# EPICS substitutions: bkhApp/Db/bkh09.substitutions
file bkhBo.db
{
pattern	{ N,       MOD,  PORT, OFF}
	{ 1, 2114-$(M), A2114,   0}
	{ 2, 2114-$(M), A2114,   1}
	{ 3, 2114-$(M), A2114,   2}
	{ 4, 2114-$(M), A2114,   3}
	{ 5, 2114-$(M), A2114,   4}
	{ 6, 2114-$(M), A2114,   5}
	{ 7, 2114-$(M), A2114,   6}
	{ 8, 2114-$(M), A2114,   7}
}
file bkhBi.db
{
pattern { N,       MOD,  PORT, OFF}
        { 1, 1104-$(M), A1104,   0}
        { 2, 1104-$(M), A1104,   1}
        { 3, 1104-$(M), A1104,   2}
        { 4, 1104-$(M), A1104,   3}
}
file bkhAdrv.db
{
pattern	{      MOD,  PORT}
	{2114-$(M), A2114}
	{1104-$(M), A1104}
}
file bkhAErr.db
{
pattern	{      MOD,  PORT}
	{1104-$(M), A1104}
}
file b9000.db{
	{ RPORT=B900R, WPORT=B900W}
}
file b9000RRegs.db
{
pattern	{ N,                 DESC,  PORT}
	{10,      "PLC Interface", B900R}
	{11, "Bus Term Diagnossi", B900R}
	{12, "Bus Coupler Status", B900R}
	{16, "anlg output length", B900R}
	{17, "anlg inputs length", B900R}
	{18, "Outpt Image length", B900R}
	{19, "Input Image length", B900R}
	{32, "Watchdog curr time", B900R}
}
file b9000WRegs.db
{
pattern	{ N,                 DESC,  PORT}
	{ 0,      "PLC Interface", B900W}
	{ 1, "Bus Term Diagnossi", B900W}
	{22,"Watchdog Tmout (ms)", B900W}
	{23,     "Watchdog Reset", B900W}
	{24,      "Watchdog type", B900W}
	{25,    "Modbus TCP mode", B900W}
}
